FUNCTION_BLOCK WAGOPEController (* Basic Function Block Type *)
  (* Standard: 61499-2 *)
  (* Version 0.2, 2003-12-04, JHC, Rockwell Automation, Renamed for better indexing. *)
  (* Compiler header: package fb.rt.wago; #include <stdio.h> *)
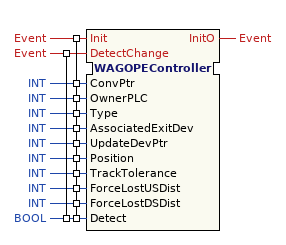
  EVENT_INPUT
    Init WITH ConvPtr, OwnerPLC, Type, AssociatedExitDev, UpdateDevPtr, Position, TrackTolerance, ForceLostUSDist, ForceLostDSDist, Detect; (* Normal Execution Request *)
    DetectChange WITH Detect; (* Normal Execution Request *)
  END_EVENT
  EVENT_OUTPUT
    InitO; (* Normal Execution Request *)
  END_EVENT
  VAR_INPUT
    ConvPtr : INT;
    OwnerPLC : INT;
    Type : INT;
    AssociatedExitDev : INT;
    UpdateDevPtr : INT;
    Position : INT;
    TrackTolerance : INT;
    ForceLostUSDist : INT;
    ForceLostDSDist : INT;
    Detect : BOOL;
  END_VAR
  VAR
    JamFault : BOOL := false;
  END_VAR
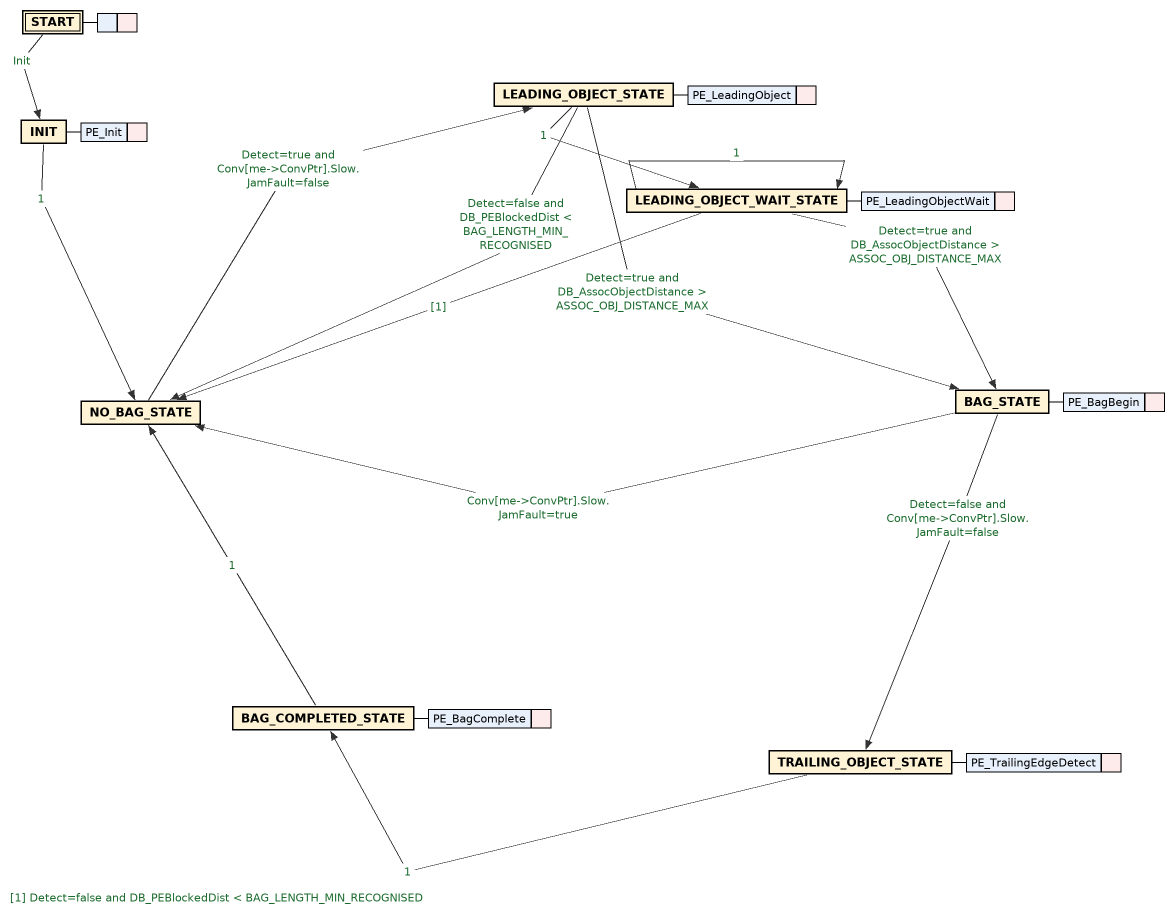
  EC_STATES
    START;
    INIT : PE_Init;
    NO_BAG_STATE;
    LEADING_OBJECT_STATE : PE_LeadingObject;
    LEADING_OBJECT_WAIT_STATE : PE_LeadingObjectWait;
    BAG_STATE : PE_BagBegin;
    TRAILING_OBJECT_STATE : PE_TrailingEdgeDetect;
    BAG_COMPLETED_STATE : PE_BagComplete;
  END_STATES
  EC_TRANSITIONS
    NO_BAG_STATE TO LEADING_OBJECT_STATE := Detect=true and Conv[me->ConvPtr].Slow.JamFault=false;
    BAG_COMPLETED_STATE TO NO_BAG_STATE := 1;
    LEADING_OBJECT_STATE TO NO_BAG_STATE := Detect=false and DB_PEBlockedDist < BAG_LENGTH_MIN_RECOGNISED;
    LEADING_OBJECT_STATE TO BAG_STATE := Detect=true and DB_AssocObjectDistance > ASSOC_OBJ_DISTANCE_MAX;
    LEADING_OBJECT_WAIT_STATE TO NO_BAG_STATE := Detect=false and DB_PEBlockedDist < BAG_LENGTH_MIN_RECOGNISED;
    LEADING_OBJECT_WAIT_STATE TO BAG_STATE := Detect=true and DB_AssocObjectDistance > ASSOC_OBJ_DISTANCE_MAX;
    BAG_STATE TO NO_BAG_STATE := Conv[me->ConvPtr].Slow.JamFault=true;
    BAG_STATE TO TRAILING_OBJECT_STATE := Detect=false and Conv[me->ConvPtr].Slow.JamFault=false;
    TRAILING_OBJECT_STATE TO BAG_COMPLETED_STATE := 1;
    START TO INIT := Init;
    INIT TO NO_BAG_STATE := 1;
    LEADING_OBJECT_STATE TO LEADING_OBJECT_WAIT_STATE := 1;
    LEADING_OBJECT_WAIT_STATE TO LEADING_OBJECT_WAIT_STATE := 1;
  END_TRANSITIONS
  ALGORITHM PE_Init IN C: (* Initialization algorithm *)
 int PosSensorID = POSSENSOR_FIRST;
 //int TempResultCode = RESULTCODE_UNKNOWNERROR;
 // 0 me->ConvPtr 24
 // 0 DevID 5

 // In Global Memory

 Conv[me->ConvPtr].Config.UpdateDev[me->UpdateDevPtr].OwnerPLC = me->OwnerPLC;
 Conv[me->ConvPtr].Config.UpdateDev[me->UpdateDevPtr].Type = me->Type;
 Conv[me->ConvPtr].Config.UpdateDev[me->UpdateDevPtr].AssociatedExitDev = me->AssociatedExitDev;

// FIND a free PosSensorID
 for(;PosSensorID < POSSENSOR_SIZE;PosSensorID++)
 {

  if( !PosSensor[PosSensorID].Slow.Enable  )
  {
   PosSensor[PosSensorID].Slow.Enable = true; // 'Allocate' it
   break;
  }
 }
 if( !PosSensor[PosSensorID].Slow.Enable  )
 {
  // Error.. No PosSensor Found
  printf("Error no valid PosSensorID(%d) found for Conv %d, Dev %d (max = %d)\n", PosSensorID, me->ConvPtr, me->UpdateDevPtr, POSSENSOR_SIZE);
  //LogErrors(UNIT_CONVEYORTRACKED,UNIT_PROCESSUPDATEDEVICESFAST,0,me->ConvPtr,me->UpdateDevPtr,PosSensorID,POSSENSOR_FIRST,PUDF_Temp,false,0,TempResultCode);
  return;
 }
 Conv[me->ConvPtr].Config.UpdateDev[me->UpdateDevPtr].PosSensorID = PosSensorID;
 Conv[me->ConvPtr].Config.UpdateDev[me->UpdateDevPtr].Pos = me->Position;
 Conv[me->ConvPtr].Config.UpdateDev[me->UpdateDevPtr].TrackTolerance = me->TrackTolerance;
 // TODO: unused... always 0
 Conv[me->ConvPtr].Config.UpdateDev[me->UpdateDevPtr].ForceLostUSDist = me->ForceLostUSDist;
 Conv[me->ConvPtr].Config.UpdateDev[me->UpdateDevPtr].ForceLostDSDist = me->ForceLostDSDist;
  END_ALGORITHM
  ALGORITHM PE_LeadingObject IN C:
  printf("PE %d on Conv %d PE_LeadingObject @ %lld\n",me->UpdateDevPtr, me->ConvPtr,Conv[me->ConvPtr].Fast.EncCount);
  DB_PosSensorID = Conv[me->ConvPtr].Config.UpdateDev[me->UpdateDevPtr].PosSensorID;
  //memcpy(&PosSensorTempFast,&PosSensor[DB_PosSensorID], sizeof(PosSensor[DB_PosSensorID])); //TODO: len = 1)

  PosSensor[DB_PosSensorID].Fast.PEBlockedEncCount = Conv[me->ConvPtr].Fast.EncCount;
  PosSensor[DB_PosSensorID].Fast.ObjectStartEncCount = PosSensor[DB_PosSensorID].Fast.PEBlockedEncCount;
  PEController_PE_LeadingObjectWait(me);
  END_ALGORITHM
  ALGORITHM PE_LeadingObjectWait IN C:

 printf("PE %d on Conv %d PE_LeadingObjectWait @ %lld\n",me->UpdateDevPtr, me->ConvPtr,Conv[me->ConvPtr].Fast.EncCount);
  DB_PosSensorID = Conv[me->ConvPtr].Config.UpdateDev[me->UpdateDevPtr].PosSensorID;
  PosSensor[DB_PosSensorID].Fast.PEClear = !(me->Detect);
  //memcpy(&PosSensorTempFast,&PosSensor[DB_PosSensorID], sizeof(PosSensor[DB_PosSensorID])); //TODO: len = 1)
 //printf("[PEC] D=%d ~D=%d !D=%d\n",me->Detect, ~(me->Detect), !(me->Detect));
 //if( (PosSensor[DB_PosSensorID].Fast.PEClear) )
  // {
    DB_AssocObjectDistance = Conv[me->ConvPtr].Fast.EncCount - PosSensor[DB_PosSensorID].Fast.ObjectStartEncCount;
    if( DB_AssocObjectDistance < ENC_COUNT_MIN )
    {
     DB_AssocObjectDistance = DB_AssocObjectDistance + ENC_COUNT_SPAN;
    }
 //printf("[PEC] %d = %d - %d\n",DB_AssocObjectDistance, Conv[me->ConvPtr].Fast.EncCount, PosSensor[DB_PosSensorID].Fast.ObjectStartEncCount);
   //}
  //else if(  !PosSensor[DB_PosSensorID].Fast.PEClear  )
   //{
    DB_PEBlockedDist = Conv[me->ConvPtr].Fast.EncCount - PosSensor[DB_PosSensorID].Fast.PEBlockedEncCount;
    if( DB_PEBlockedDist < ENC_COUNT_MIN )
    {
     DB_PEBlockedDist = DB_PEBlockedDist + ENC_COUNT_SPAN;
    }

   //}
  END_ALGORITHM
  ALGORITHM PE_BagBegin IN C:
  printf("PE %d on Conv %d PE_BagBegin @ EC %lld, BagDSEC = %lld\n",me->UpdateDevPtr, me->ConvPtr,Conv[me->ConvPtr].Fast.EncCount, PosSensor[DB_PosSensorID].Fast.PEBlockedEncCount);
  DB_PosSensorID = Conv[me->ConvPtr].Config.UpdateDev[me->UpdateDevPtr].PosSensorID;
  //memcpy(&PosSensorTempFast,&PosSensor[DB_PosSensorID], sizeof(PosSensor[DB_PosSensorID])); //TODO: len = 1)


  //"<BAG STATE> ACTIONS"

 PosSensor[DB_PosSensorID].Fast.AssObjDSEncCount = PosSensor[DB_PosSensorID].Fast.ObjectStartEncCount;
 PosSensor[DB_PosSensorID].Fast.BagDSEncCount = PosSensor[DB_PosSensorID].Fast.PEBlockedEncCount;

 //"INCREMENT THE QUEUE WRITE POINTER"

 DB_WritePtr = BagPositionEventQueue.WritePtr;
 DB_WritePtr = DB_WritePtr + 1;
 if( DB_WritePtr >= BagPositionEventQueue.QUEUE_SIZE )
 {
  DB_WritePtr = BagPositionEventQueue.QUEUE_FIRST;
 }

 //"INCREMENT THE UPDATE SEQUENCE NUMBER"

 BagPositionEventQueue.MasterSequenceNumber = BagPositionEventQueue.MasterSequenceNumber + 1;
 if( BagPositionEventQueue.MasterSequenceNumber >= QUEUESEQUENCENUMBER_SIZE )
 {
  BagPositionEventQueue.MasterSequenceNumber = QUEUESEQUENCENUMBER_FIRST;
 }

 //"UPDATE THE QUEUE DATA"

 BagPositionEventQueue.Data[DB_WritePtr].TimeStamp = TimeSinceMidnight_ms;
 BagPositionEventQueue.Data[DB_WritePtr].EventType = BAGPOSITIONEVENTTYPE_DSUPDATE;
 BagPositionEventQueue.Data[DB_WritePtr].Update.ConvID = me->ConvPtr;
 BagPositionEventQueue.Data[DB_WritePtr].Update.UpdateDevID = me->UpdateDevPtr;
 BagPositionEventQueue.Data[DB_WritePtr].Update.BagID = BAGID_NONE;
 BagPositionEventQueue.Data[DB_WritePtr].Update.BagDSEncCount = PosSensor[DB_PosSensorID].Fast.BagDSEncCount;
 BagPositionEventQueue.Data[DB_WritePtr].Update.BagUSEncCount = NO_DATA;
 BagPositionEventQueue.Data[DB_WritePtr].Update.BagUSEncCountOnDSConv = NO_DATA;
 BagPositionEventQueue.Data[DB_WritePtr].SequenceNumber = BagPositionEventQueue.MasterSequenceNumber;
 BagPositionEventQueue.WritePtr = DB_WritePtr;
 PEController_PE_PrintBagPositionEventQueue(me);
  END_ALGORITHM
  ALGORITHM PE_TrailingEdgeDetect IN C:
 printf("PE %d on Conv %d Trailing edge PEUnblockedEncCount = %lld\n",me->UpdateDevPtr, me->ConvPtr,Conv[me->ConvPtr].Fast.EncCount);
 DB_PosSensorID = Conv[me->ConvPtr].Config.UpdateDev[me->UpdateDevPtr].PosSensorID;
 PUDF_DSConvPtr = Conv[me->ConvPtr].Config.ExitDev[EXITDEVICE_MOST_DOWNSTREAM].EntryConvID;
 //memcpy(&PosSensorTempFast,&PosSensor[DB_PosSensorID], sizeof(PosSensor[DB_PosSensorID])); //TODO: len = 1)
 PosSensor[DB_PosSensorID].Fast.PEUnblockedEncCount = Conv[me->ConvPtr].Fast.EncCount;
 PosSensor[DB_PosSensorID].Fast.BagUSEncCount = Conv[me->ConvPtr].Fast.EncCount;
 PosSensor[DB_PosSensorID].Fast.BagUSEncCountOnDSConv = Conv[PUDF_DSConvPtr].Fast.EncCount;
  END_ALGORITHM
  ALGORITHM PE_BagComplete IN C:
 printf("PE %d on Conv %d PEController_PE_BagComplete @ %lld\n",me->UpdateDevPtr, me->ConvPtr,PosSensor[DB_PosSensorID].Fast.PEUnblockedEncCount);
  DB_PosSensorID = Conv[me->ConvPtr].Config.UpdateDev[me->UpdateDevPtr].PosSensorID;
  //memcpy(&PosSensorTempFast,&PosSensor[DB_PosSensorID], sizeof(PosSensor[DB_PosSensorID])); //TODO: len = 1)
 /*
 "ON ENTRY FROM <TRAILING OBJECT> STATE WITHOUT FAULT$N"
 "Store the associated object upstream encoder count"
 */

 PosSensor[DB_PosSensorID].Fast.AssObjUSEncCount = PosSensor[DB_PosSensorID].Fast.PEUnblockedEncCount;

 //"INCREMENT THE QUEUE WRITE POINTER"

 DB_WritePtr = BagPositionEventQueue.WritePtr;
 DB_WritePtr = DB_WritePtr + 1;
 if( DB_WritePtr >= BagPositionEventQueue.QUEUE_SIZE )
 {
  DB_WritePtr = BagPositionEventQueue.QUEUE_FIRST;
 }

 //"INCREMENT THE UPDATE SEQUENCE NUMBER"

 BagPositionEventQueue.MasterSequenceNumber = BagPositionEventQueue.MasterSequenceNumber + 1;
 if( BagPositionEventQueue.MasterSequenceNumber >= QUEUESEQUENCENUMBER_SIZE )
 {
  BagPositionEventQueue.MasterSequenceNumber = QUEUESEQUENCENUMBER_FIRST;
 }

 //"UPDATE THE QUEUE DATA"

 BagPositionEventQueue.Data[DB_WritePtr].TimeStamp = TimeSinceMidnight_ms;
 BagPositionEventQueue.Data[DB_WritePtr].EventType = BAGPOSITIONEVENTTYPE_USUPDATE;
 BagPositionEventQueue.Data[DB_WritePtr].Update.ConvID = me->ConvPtr;
 BagPositionEventQueue.Data[DB_WritePtr].Update.UpdateDevID = me->UpdateDevPtr;
 BagPositionEventQueue.Data[DB_WritePtr].Update.BagID = Conv[me->ConvPtr].Slow.UpdateDev[me->UpdateDevPtr].LastUpdateBagID;
 BagPositionEventQueue.Data[DB_WritePtr].Update.BagDSEncCount = NO_DATA;
 BagPositionEventQueue.Data[DB_WritePtr].Update.BagUSEncCount = PosSensor[DB_PosSensorID].Fast.BagUSEncCount;
 BagPositionEventQueue.Data[DB_WritePtr].Update.BagUSEncCountOnDSConv = PosSensor[DB_PosSensorID].Fast.BagUSEncCountOnDSConv;
 BagPositionEventQueue.Data[DB_WritePtr].SequenceNumber = BagPositionEventQueue.MasterSequenceNumber;
 BagPositionEventQueue.WritePtr = DB_WritePtr;
 PEController_PE_PrintBagPositionEventQueue(me);
  END_ALGORITHM
  ALGORITHM PE_PrintBagPositionEventQueue IN C:
 printf("PEController_PE_PrintBagPositionEventQueue: %d vs %d\n", BagPositionEventQueue.ReadPtr, BagPositionEventQueue.WritePtr);
 int queueIndex = BagPositionEventQueue.ReadPtr;
 int endIndex = BagPositionEventQueue.WritePtr;
 //while( queueIndex < endIndex )
 //{
  printf("Time: %d, Type %d, ConvID %d, DevID %d, BagID %d, DSEC %d, USEC %d, USEConDSConv %d, SeqNum %d\n",
   BagPositionEventQueue.Data[queueIndex].TimeStamp,
   BagPositionEventQueue.Data[queueIndex].EventType,
   BagPositionEventQueue.Data[queueIndex].Update.ConvID,
   BagPositionEventQueue.Data[queueIndex].Update.UpdateDevID,
   BagPositionEventQueue.Data[queueIndex].Update.BagID,
   BagPositionEventQueue.Data[queueIndex].Update.BagDSEncCount,
   BagPositionEventQueue.Data[queueIndex].Update.BagUSEncCount,
   BagPositionEventQueue.Data[queueIndex].Update.BagUSEncCountOnDSConv,
   BagPositionEventQueue.Data[queueIndex].SequenceNumber
  );
  queueIndex++;
 //}
  END_ALGORITHM
END_FUNCTION_BLOCK
